(* CoDeSys 2.3.9.28 project: Automatic_Water_Tank.pro *)
(* Libraries: Standard.lib 4.10.05 11:14:46, IecSfc.lib 13.4.06 14:51:28, SYSLIBCALLBACK.LIB 26.9.08 15:43:52 *)

(* POU PLC_PRG, LD *)
PROGRAM PLC_PRG
VAR
	start: BOOL;
	C1: BOOL;
	MV1: BOOL;
	MV2: BOOL;
	HEATER: BOOL;
	MOTOR: BOOL;
	Name: BOOL;

	T1: TON;
	V1: TIME;
	TIM1: BOOL;

	SENSOR1: BOOL;
	SENSOR2: BOOL;
	SENSOR3: BOOL;
	ref: INT:=90;
	tempt: INT;

	CTU1: CTU;
	cv1: INT;

END_VAR
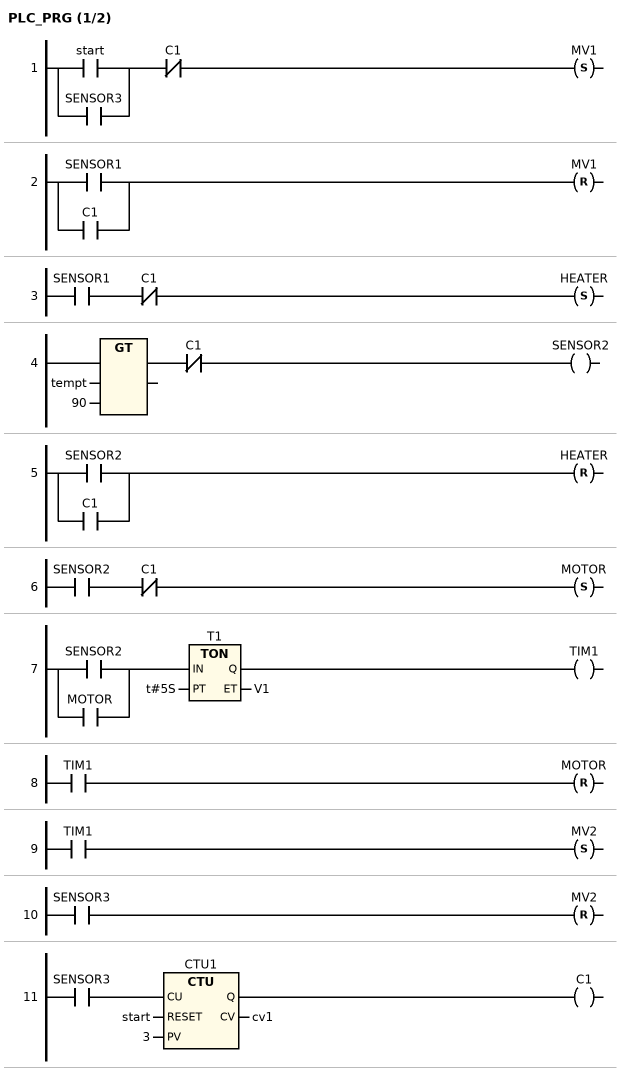
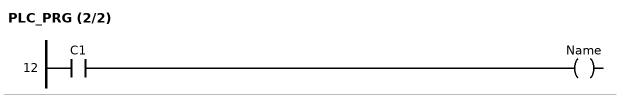
_LD_ (* Ladder Diagram *)
NETWORK 1
	{ [start] | [SENSOR3] } - [/C1] --- (S MV1)
NETWORK 2
	{ [SENSOR1] | [C1] } --- (R MV1)
NETWORK 3
	[SENSOR1] - [/C1] --- (S HEATER)
NETWORK 4
	GT(tempt, 90) - [/C1] --- (SENSOR2)
NETWORK 5
	{ [SENSOR2] | [C1] } --- (R HEATER)
NETWORK 6
	[SENSOR2] - [/C1] --- (S MOTOR)
NETWORK 7
	{ [SENSOR2] | [MOTOR] } - T1:TON(IN: *, PT: t#5S, ET => V1) --- (TIM1)
NETWORK 8
	[TIM1] --- (R MOTOR)
NETWORK 9
	[TIM1] --- (S MV2)
NETWORK 10
	[SENSOR3] --- (R MV2)
NETWORK 11
	[SENSOR3] - CTU1:CTU(CU: *, RESET: start, PV: 3, CV => cv1) --- (C1)
NETWORK 12
	[C1] --- (Name)
_END_LD_
(* the same logic as Structured Text *)
(* Network 1 *)
IF (start OR SENSOR3) AND NOT C1 THEN MV1 := TRUE; END_IF;
(* Network 2 *)
IF SENSOR1 OR C1 THEN MV1 := FALSE; END_IF;
(* Network 3 *)
IF SENSOR1 AND NOT C1 THEN HEATER := TRUE; END_IF;
(* Network 4: see the listing above *)
(* Network 5 *)
IF SENSOR2 OR C1 THEN HEATER := FALSE; END_IF;
(* Network 6 *)
IF SENSOR2 AND NOT C1 THEN MOTOR := TRUE; END_IF;
(* Network 7 *)
T1(IN := SENSOR2 OR MOTOR, PT := t#5S);
V1 := T1.ET;
TIM1 := T1.Q;
(* Network 8 *)
IF TIM1 THEN MOTOR := FALSE; END_IF;
(* Network 9 *)
IF TIM1 THEN MV2 := TRUE; END_IF;
(* Network 10 *)
IF SENSOR3 THEN MV2 := FALSE; END_IF;
(* Network 11 *)
CTU1(CU := SENSOR3, RESET := start, PV := 3);
cv1 := CTU1.CV;
C1 := CTU1.Q;
(* Network 12 *)
Name := C1;
END_PROGRAM

(* Visualisation BLE
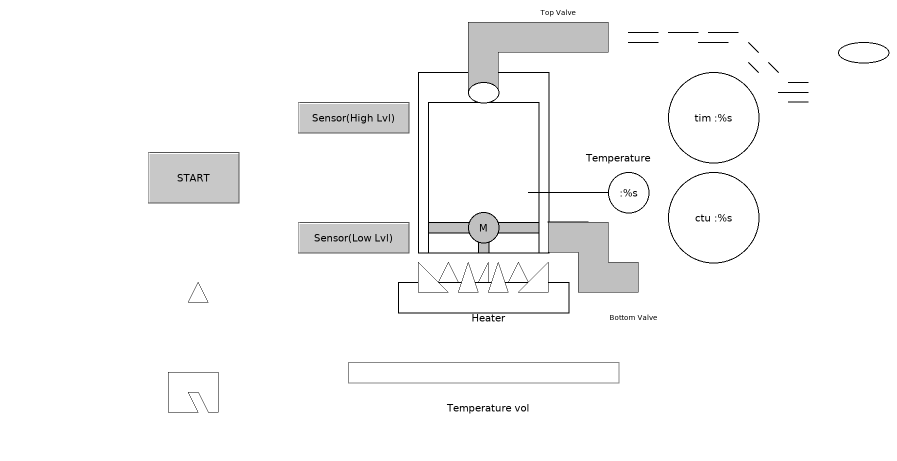
ellipse at (850,50)-(901,71): alarm colour if PLC_PRG.MV1
rounded rectangle at (440,110)-(551,261): alarm colour if PLC_PRG.HEATER
button at (160,160)-(251,211): text "START"; taps PLC_PRG.start
button at (310,110)-(421,141): text "Sensor(High Lvl)"; taps PLC_PRG.SENSOR1
ellipse at (680,180)-(771,271): text "ctu :%s"; shows PLC_PRG.cv1; alarm colour if PLC_PRG.cv1
button at (310,230)-(421,261): text "Sensor(Low Lvl)"; taps PLC_PRG.SENSOR3
ellipse at (680,80)-(771,171): text "tim :%s"; shows PLC_PRG.T1.ET; alarm colour if PLC_PRG.T1.ET
rectangle at (410,290)-(581,321): alarm colour if PLC_PRG.HEATER
polygon at (530,270)-(560,300): alarm colour if PLC_PRG.HEATER
polygon at (430,270)-(460,300): alarm colour if PLC_PRG.HEATER
polygon at (500,270)-(520,300): alarm colour if PLC_PRG.HEATER
polygon at (470,270)-(490,300): alarm colour if PLC_PRG.HEATER
ellipse at (620,180)-(661,221): text ":%s"; shows PLC_PRG.tempt; alarm colour if PLC_PRG.tempt
polygon at (450,270)-(470,290): alarm colour if PLC_PRG.HEATER
polygon at (490,270)-(500,290): alarm colour if PLC_PRG.HEATER
polygon at (520,270)-(540,290): alarm colour if PLC_PRG.HEATER
rectangle at (480,130)-(491,151): alarm colour if PLC_PRG.MV1
rectangle at (500,130)-(511,151): alarm colour if PLC_PRG.MV1
rectangle at (480,160)-(491,181): alarm colour if PLC_PRG.MV1
rectangle at (500,160)-(511,181): alarm colour if PLC_PRG.MV1
rectangle at (490,190)-(501,211): alarm colour if PLC_PRG.MV1
rounded rectangle at (440,120)-(551,261): alarm colour if PLC_PRG.MOTOR
rectangle at (660,270)-(691,281): alarm colour if PLC_PRG.MV2
rectangle at (660,290)-(691,301): alarm colour if PLC_PRG.MV2
rectangle at (700,280)-(731,291): alarm colour if PLC_PRG.MV2
rectangle at (740,290)-(771,301): alarm colour if PLC_PRG.MV2
ellipse at (450,130)-(541,141): alarm colour if PLC_PRG.MOTOR
ellipse at (460,150)-(531,161): alarm colour if PLC_PRG.MOTOR
ellipse at (470,170)-(521,181): alarm colour if PLC_PRG.MOTOR
ellipse at (480,190)-(511,201): alarm colour if PLC_PRG.MOTOR
ellipse at (490,210)-(501,221): alarm colour if PLC_PRG.MOTOR
rectangle at (440,200)-(561,261): alarm colour if PLC_PRG.MV2
rectangle at (490,230)-(501,261): alarm colour if PLC_PRG.MOTOR
rectangle at (440,230)-(491,241): alarm colour if PLC_PRG.MOTOR
rectangle at (500,230)-(551,241): alarm colour if PLC_PRG.MOTOR
ellipse at (480,220)-(511,251): text "M"; alarm colour if PLC_PRG.MOTOR
rectangle at (580,150)-(681,181): text "Temperature"
rectangle at (520,10)-(621,31): text "Top Valve"
rectangle at (590,310)-(701,341): text "Bottom Valve"
rectangle at (450,320)-(551,331): text "Heater"
rectangle at (430,400)-(571,431): text "Temperature vol"
rectangle at (850,70)-(901,141): alarm colour if PLC_PRG.MV1
rounded rectangle at (840,140)-(911,151): alarm colour if PLC_PRG.MV1
rounded rectangle at (830,150)-(921,161): alarm colour if PLC_PRG.MV1
rectangle at (900,90)-(911,111): alarm colour if PLC_PRG.MV1
rectangle at (840,90)-(851,111): alarm colour if PLC_PRG.MV1
rectangle at (910,80)-(921,121): alarm colour if PLC_PRG.MV1
rectangle at (830,80)-(841,121): alarm colour if PLC_PRG.MV1
rounded rectangle at (840,60)-(911,71): alarm colour if PLC_PRG.MV1
rectangle at (870,40)-(881,51): alarm colour if PLC_PRG.MV1
ellipse at (860,90)-(891,121): alarm colour if PLC_PRG.MV1
ellipse at (630,30)-(641,41): alarm colour if PLC_PRG.MV1
polygon at (20,270)-(100,350): alarm colour if PLC_PRG.Name
polygon at (110,270)-(170,350): alarm colour if PLC_PRG.Name
polygon at (180,270)-(240,350): alarm colour if PLC_PRG.Name
polygon at (250,270)-(320,350): alarm colour if PLC_PRG.Name
polygon at (330,270)-(390,350): alarm colour if PLC_PRG.Name
polygon at (160,360)-(250,460): alarm colour if PLC_PRG.Name
ellipse at (260,430)-(281,451): alarm colour if PLC_PRG.Name
polygon at (620,20)-(830,120): alarm colour if PLC_PRG.MV1
polyline at (640,40)-(670,40): alarm colour if PLC_PRG.MV1
polyline at (640,50)-(670,50): alarm colour if PLC_PRG.MV1
polyline at (680,40)-(710,40): alarm colour if PLC_PRG.MV1
polyline at (800,90)-(820,90): alarm colour if PLC_PRG.MV1
polyline at (790,100)-(820,100): alarm colour if PLC_PRG.MV1
polyline at (800,110)-(820,110): alarm colour if PLC_PRG.MV1
polyline at (780,70)-(790,80): alarm colour if PLC_PRG.MV1
polyline at (760,70)-(770,80): alarm colour if PLC_PRG.MV1
polyline at (710,50)-(740,50): alarm colour if PLC_PRG.MV1
polyline at (720,40)-(750,40): alarm colour if PLC_PRG.MV1
polyline at (760,50)-(770,60): alarm colour if PLC_PRG.MV1
polygon at (480,30)-(620,100): alarm colour if PLC_PRG.MV1
ellipse at (480,90)-(511,111): alarm colour if PLC_PRG.MV1
polygon at (560,230)-(650,300): alarm colour if PLC_PRG.MV2
6 more shapes without text or variables
*)
